PROGRAM POU_TEST
VAR
	
TEST	:fb_OrdreAllumage_3; 
END_VAR

TEST(
	Objet:= , 
	iNbreObjet_A_Allumer:= , 
	sOrdreDePriorite:= , 
	bOptimisationOrdreAllumage:= , 
	iNbreObjetAllume=> , 
	sPrioriteActuelle=> , 
	bError=> , 
	sError=> );

END_PROGRAM

(* stored: Version 1.1.0.1, ProductVersion 3.1.4024.12
   POU POU_TEST: Id {6c244330-7fc7-42cb-962c-460bb006b5ae}, SpecialFunc None *)
